PROGRAM MAIN
VAR
	testFB : TestFB;
	monitoredValueUpdate : MonitoredValueUpdate;
	main_state : MAIN_ST := MAIN_ST.STARTUP;
	hmi_FB   : HMI_FB;
	
	//main variables 
	bInputError : BOOL := FALSE;
END_VAR

//Always run the function blocks
testFB();
monitoredValueUpdate();
hmi_FB();

IF NOT gIO.DI_ESTOP_L2 THEN
	main_state := MAIN_ST.ESTOP;
END_IF

CASE MAIN_STATE OF 
	MAIN_ST.STARTUP: 
		testFB(command_StartTest:=FALSE, command_StopTest:=FALSE,command_Reset:=FALSE);
		monitoredValueUpdate(resetDefaults:=TRUE);
		main_state := MAIN_ST.IDLE;
	MAIN_ST.IDLE:
		IF gHMI.bStartButtonState THEN
			gHMI.bStartButtonState := FALSE;
			main_state := MAIN_ST.TESTING;
			testFB(command_StartTest:=TRUE, bNoMethane:=NOT gHMI.bMethaneCheckBox);
		END_IF
	MAIN_ST.TESTING:
		IF gHMI.bStopButtonState THEN
			gHMI.bStopButtonState := FALSE;
			testFB(command_StopTest:=TRUE);
		END_IF
		IF gHMI.bStartSeedButtonState AND NOT testFB.bSeedInhibit THEN
			gHMI.bStartSeedButtonState := FALSE;
			testFB(command_StartSeed := TRUE);
		END_IF
		IF gMachine.testCell.state = TEST_STATE.COMPLETE 
			OR gMachine.testCell.state = TEST_STATE.STOP
			OR gMachine.testCell.state = TEST_STATE.ESTOP THEN
				main_state := MAIN_ST.IDLE;
		END_IF
	MAIN_ST.ESTOP:
		gMachine.testCell.state := TEST_STATE.ESTOP;
		IF gIO.DI_ESTOP_L2 THEN
			gMachine.testCell.state := TEST_STATE.WAIT_FOR_RESET;
			main_state := MAIN_ST.WAIT_FOR_RESET;
			
		END_IF
	MAIN_ST.WAIT_FOR_RESET:
		IF gHMI.bReset THEN
			gHMI.bReset := FALSE;
			testFB(command_Reset:=TRUE);
			main_state := MAIN_ST.RESETTING;
		END_IF
	MAIN_ST.RESETTING:
		IF gMachine.testCell.state = TEST_STATE.IDLE THEN
			main_state := MAIN_ST.IDLE;
		END_IF	
END_CASE

gHMI.bEStopPressed := NOT gIO.DI_24VAtSolenoids;

END_PROGRAM

(* stored: Version 1.1.0.1, ProductVersion 3.1.4024.12
   POU MAIN: Id {95f0d3d7-ef12-463a-a495-742fe761b35c}, SpecialFunc None *)
